PROGRAM Config_Slow
VAR
	//temp					:INT;
	//temp_load				:INT :=1;
	//temp_save				:INT :=0;
	Once					:BOOL :=TRUE;
	juan					:INT;
	//saving_config			:BOOL :=FALSE;
	//config_status			:BOOL :=FALSE;
	config_count			:INT;		
END_VAR


IF Clock.DateTimeInitialised THEN
	
	FOR juan := 1 TO config_speed DO
		Config.Update();
	END_FOR

	
	
	load_config();
	
	IF config.Initialised() THEN
		save_config();	
	END_IF

END_IF

METHOD load_config : BOOL
VAR_INPUT
END_VAR
(*//IF once =TRUE THEN
	IF Config.Initialised(temp_load) = FALSE THEN
		Config.Update(temp_load);


	ELSIF temp_load = 11 THEN
		Message:='Data Loaded';
		Once:=FALSE;
	ELSE
		Config.Update(temp_load);
		Config.Update(temp_load);
		temp_load:=temp_load+1;
	END_IF
//END_IF
*)	
//2500
//Config.Update(1);
//Config.Update(2);
//Config.Update(3);
//Config.Update(4);
//Config.Update(5);
//Config.Update(6);
//Config.Update(7);
//Config.Update(8);
//Config.Update(9);
//Config.Update(10);
//Config.Update(11);

IF once AND config.Initialised() THEN
	once:=FALSE;
	IF language.english THEN
		Message:='Data loaded';
	ELSE
		Message:='Dados carregados';
	END_IF
END_IF


(*
IF config_count = 1000 THEN
	config_count:=0;
	IF temp_load = 11 THEN
		temp_load:=0;
	END_IF 
	temp_load:=temp_load+1;
END_IF
*)
END_METHOD

METHOD save_config : BOOL
VAR_INPUT
END_VAR

	
IF Config_Request= TRUE THEN
	Config_Request:=FALSE;

	config_count:=0;
	//temp_save:=temp_save+1;
		
END_IF

config_count:=config_count+config_speed;

IF config_count > 7000 THEN
	config_count := 0;
	IF configuring THEN
		Message:=Config_Message;
		configuring:=FALSE;
	END_IF
	
END_IF
END_METHOD

END_PROGRAM

(* stored: Version 1.1.0.1, ProductVersion 3.1.4020.12
   POU Config_Slow: Id {68820ce0-f190-48fe-919d-63c0e6e8e6eb}, SpecialFunc None
   Method load_config: Id {097443b6-b1ac-4abf-8692-1b8c84698695}
   Method save_config: Id {ede5b518-086f-4687-bb4d-0480b77911be} *)
